// Mitsubishi GX Works2 project: Falling_pulse_Not_use_PULSE   PLC: Q03UDV

PROGRAM MAIN
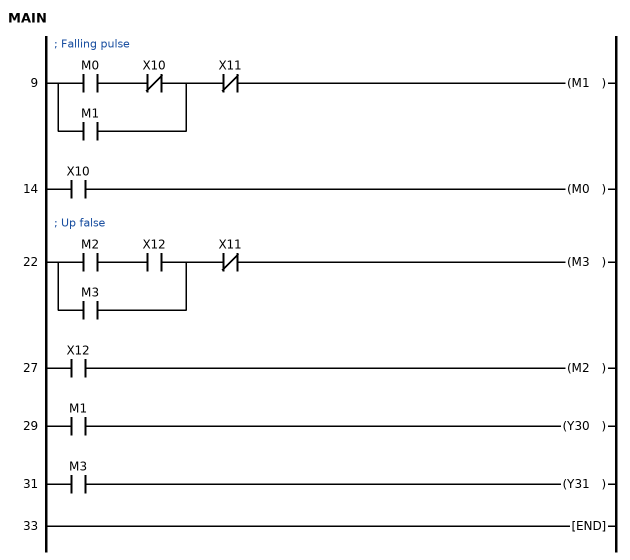
; Falling pulse
9     LD      M0
      ANI     X10
      OR      M1
      ANI     X11
      OUT     M1
14    LD      X10
      OUT     M0
; Up false
22    LD      M2
      AND     X12
      OR      M3
      ANI     X11
      OUT     M3
27    LD      X12
      OUT     M2
29    LD      M1
      OUT     Y30
31    LD      M3
      OUT     Y31
33    END
END_PROGRAM
